FUNCTION_BLOCK FB_HomingProcessor
VAR_IN_OUT
	J1, J2, J3, J4, J5, J6: AXIS_REF;
	AxisGroup: AXIS_GROUP_REF_SM3;
	GroupHandler: FB_GroupHandler;
	Controller: FB_Controller;
END_VAR

VAR_INPUT
	J1_Limit, J2_Limit, J3_Limit, J4_Limit, J5_Limit, J6_Limit: BOOL;
	Enable: BOOL;
	Reset: BOOL;
	StoredPositions: REFERENCE TO ARRAY[GVL.POS_ARR_BEG..GVL.POS_ARR_END] OF DUT_StoredPosition;
	VisionRegisters: REFERENCE TO ARRAY[GVL.VIS_ARR_BEG..GVL.VIS_ARR_END] OF DUT_VisionRegister;
	Flags: REFERENCE TO ARRAY[GVL.FLG_ARR_BEG..GVL.FLG_ARR_END] OF DUT_Flags;
END_VAR
VAR_OUTPUT
	Done: BOOL;
	Busy: BOOL;
	Error: BOOL;
	ErrorID: UDINT;
END_VAR
VAR
	_ExecuteRtrig: R_TRIG;
	_ExecuteFtrig: F_TRIG;
	_ResetRtrig: R_TRIG;
	_ErrorRtrig: R_TRIG;
	
	_SequenceMain: INT;
	_StartHoming: BOOL;
	
	_SMC_Homing_J1, _SMC_Homing_J2, _SMC_Homing_J3: MC_Home;
	_SMC_Homing_J4, _SMC_Homing_J5, _SMC_Homing_J6: MC_Home;
    _ST_HomingOptions_J1,_ST_HomingOptions_J2,_ST_HomingOptions_J3: ST_HomingOptions;
    _ST_HomingOptions_J4,_ST_HomingOptions_J5,_ST_HomingOptions_J6: ST_HomingOptions;
	
	_MC_SetPosition_J1, _MC_SetPosition_J2, _MC_SetPosition_J3: MC_SetPosition;
	_MC_SetPosition_J4, _MC_SetPosition_J5, _MC_SetPosition_J6: MC_SetPosition;
    _ST_SetPositionsOptions_J1,_ST_SetPositionsOptions_J2,_ST_SetPositionsOptions_J3: ST_SetPositionOptions;
    _ST_SetPositionsOptions_J4,_ST_SetPositionsOptions_J5,_ST_SetPositionsOptions_J6: ST_SetPositionOptions;
	
	_HomingVelocityFast: LREAL:= 10.0;
	_HomingVelocitySlow: LREAL:= 5.0;
	_HomingVelocitySlowSlow: LREAL:= 1.0;
	_HomingAcceleration: LREAL:= 1000.0;
	_HomingJerk: LREAL:= 10000.0;
	
	_MoveToPose: BOOL;
	_MoveCommand: ST_MoveCmd;
	_MoveCommandProcessor: MoveCmdProcessor;
	
	_i, _j, _k: INT;
	_FirstScan: BOOL:=TRUE;
END_VAR

VAR CONSTANT
	STEP_DONE: 					INT := 9999;
	STEP_IDLE: 					INT := 0000;
	STEP_GROUP_ENABLE: 			INT := 0030;
	STEP_WAIT_ENABLE: 			INT := 0035;
	STEP_FAST_HOME_G1:			INT := 0040;
	STEP_WAIT_FAST_HOME_G1:		INT := 0045;
	STEP_SLOW_HOME_G1:			INT := 0050;
	STEP_WAIT_SLOW_HOME_G1:		INT := 0055;
	
	STEP_FAST_HOME_G2:			INT := 0060;
	STEP_WAIT_FAST_HOME_G2:		INT := 0065;
	STEP_SLOW_HOME_G2:			INT := 0070;
	STEP_WAIT_SLOW_HOME_G2:		INT := 0075;
	
	STEP_FAST_HOME_G3:			INT := 0080;
	STEP_WAIT_FAST_HOME_G3:		INT := 0085;
	STEP_SLOW_HOME_G3:			INT := 0090;
	STEP_WAIT_SLOW_HOME_G3:		INT := 0095;
	
	STEP_MOVE_TO_POSE:			INT := 1000;
	STEP_WAIT_MOVE_TO_POSE:		INT := 1010;
	STEP_WAIT_POSE_DONE:		INT := 1020;
END_VAR

_ExecuteRtrig(CLK:=);
_ExecuteFtrig(CLK:=);
_ResetRtrig(CLK:=Reset);

IF _FirstScan THEN
	//
END_IF

CASE _SequenceMain OF
	STEP_DONE: // done
		Busy := FALSE;
		Done := TRUE;
		_MoveCommandProcessor.M_Home();
		_SequenceMain := STEP_IDLE;
		
		_SMC_Homing_J1.Execute := FALSE;
		_SMC_Homing_J2.Execute := FALSE;
		_SMC_Homing_J3.Execute := FALSE;
		_SMC_Homing_J4.Execute := FALSE;
		_SMC_Homing_J5.Execute := FALSE;
		_SMC_Homing_J6.Execute := FALSE;
		(*J1.bSWLimitEnable := TRUE;
		J2.bSWLimitEnable := TRUE;
		J3.bSWLimitEnable := TRUE;
		J4.bSWLimitEnable := TRUE;
		J5.bSWLimitEnable := TRUE;
		J6.bSWLimitEnable := TRUE;*)
		
	STEP_IDLE: // IDLE
		IF _StartHoming AND Enable THEN
			_StartHoming := FALSE;
			Busy := TRUE;
			Done := FALSE;
			_SequenceMain := STEP_GROUP_ENABLE;
			Flags[GVL.HOME_COMPLETE].Value := FALSE;
		END_IF
		
	STEP_GROUP_ENABLE:
		IF GroupHandler.M_EnableGroup() THEN
			_SequenceMain := STEP_WAIT_ENABLE;
		ELSE
			_SequenceMain := STEP_DONE;
			Error := TRUE;
			ErrorID := GroupHandler.ErrorID;
		END_IF
		
	STEP_WAIT_ENABLE:
		// TODO add timeout timer here
		IF GroupHandler.P_GroupEnabled THEN
			_SequenceMain := STEP_FAST_HOME_G1;
		END_IF;
		
	STEP_FAST_HOME_G1:	
		_SMC_Homing_J1.Execute := TRUE;
		_SMC_Homing_J2.Execute := TRUE;
		_SMC_Homing_J3.Execute := TRUE;
		//_SMC_Homing_J1.bReturnToZero := FALSE;
		//_SMC_Homing_J2.bReturnToZero := FALSE;
		//_SMC_Homing_J3.bReturnToZero := FALSE;
		_SMC_Homing_J1.Options.SearchVelocity := _HomingVelocitySlow;
		_SMC_Homing_J2.Options.SearchVelocity := _HomingVelocitySlow;
		_SMC_Homing_J3.Options.SearchVelocity := _HomingVelocitySlow;
		//J1.bSWLimitEnable := FALSE;
		//J2.bSWLimitEnable := FALSE;
		//J3.bSWLimitEnable := FALSE;
		_SequenceMain := STEP_WAIT_FAST_HOME_G1;
		
	STEP_WAIT_FAST_HOME_G1: // wait fast home group 1
		IF _SMC_Homing_J1.Done
			AND _SMC_Homing_J2.Done
			AND _SMC_Homing_J3.Done THEN
				_SMC_Homing_J1.Execute := FALSE;
				_SMC_Homing_J2.Execute := FALSE;
				_SMC_Homing_J3.Execute := FALSE;
				_SequenceMain := STEP_SLOW_HOME_G1;
		END_IF
		
	STEP_SLOW_HOME_G1: // slow home group 1
		_SMC_Homing_J1.Execute := TRUE;
		_SMC_Homing_J2.Execute := TRUE;
		_SMC_Homing_J3.Execute := TRUE;
		//_SMC_Homing_J1.bReturnToZero := TRUE;
		//_SMC_Homing_J2.bReturnToZero := TRUE;
		//_SMC_Homing_J3.bReturnToZero := TRUE;
		_SMC_Homing_J1.Options.SearchVelocity := _HomingVelocitySlowSlow;
		_SMC_Homing_J2.Options.SearchVelocity := _HomingVelocitySlowSlow;
		_SMC_Homing_J3.Options.SearchVelocity := _HomingVelocitySlowSlow;
		_SequenceMain := STEP_WAIT_SLOW_HOME_G1;
		
	STEP_WAIT_SLOW_HOME_G1:
		IF _SMC_Homing_J1.Done
			AND _SMC_Homing_J2.Done
			AND _SMC_Homing_J3.Done THEN
				_SMC_Homing_J1.Execute := FALSE;
				_SMC_Homing_J2.Execute := FALSE;
				_SMC_Homing_J3.Execute := FALSE;
				_SequenceMain := STEP_FAST_HOME_G2;
		END_IF
		
	STEP_FAST_HOME_G2:		
		_SMC_Homing_J4.Execute := TRUE;
		_SMC_Homing_J5.Execute := TRUE;
		//_SMC_Homing_J4.bReturnToZero := FALSE;
		//_SMC_Homing_J5.bReturnToZero := FALSE;
		_SMC_Homing_J4.Options.SearchVelocity := _HomingVelocitySlow;
		_SMC_Homing_J5.Options.SearchVelocity := _HomingVelocitySlow;
		//J4.bSWLimitEnable := FALSE;
		//J5.bSWLimitEnable := FALSE;
		_SequenceMain := STEP_WAIT_FAST_HOME_G2;
		
	STEP_WAIT_FAST_HOME_G2:
		IF _SMC_Homing_J4.Done
			AND _SMC_Homing_J5.Done THEN
				_SMC_Homing_J4.Execute := FALSE;
				_SMC_Homing_J5.Execute := FALSE;
				_SequenceMain := STEP_SLOW_HOME_G2;
		END_IF
		
	STEP_SLOW_HOME_G2:
		_SMC_Homing_J4.Execute := TRUE;
		_SMC_Homing_J5.Execute := TRUE;
		//_SMC_Homing_J4.bReturnToZero := TRUE;
		//_SMC_Homing_J5.bReturnToZero := TRUE;
		_SMC_Homing_J4.Options.SearchVelocity := _HomingVelocitySlowSlow;
		_SMC_Homing_J5.Options.SearchVelocity := _HomingVelocitySlowSlow;
		_SequenceMain := STEP_WAIT_SLOW_HOME_G2;
		
	STEP_WAIT_SLOW_HOME_G2:
		IF _SMC_Homing_J4.Done
			AND _SMC_Homing_J5.Done THEN
				_SMC_Homing_J4.Execute := FALSE;
				_SMC_Homing_J5.Execute := FALSE;
				_SequenceMain := STEP_FAST_HOME_G3;
		END_IF
		
	STEP_FAST_HOME_G3:
		_SMC_Homing_J6.Execute := TRUE;
		//_SMC_Homing_J6.bReturnToZero := FALSE;
		_SMC_Homing_J6.Options.SearchVelocity := _HomingVelocitySlow;
		//J6.bSWLimitEnable := FALSE;
		_SequenceMain := STEP_WAIT_FAST_HOME_G3;
		
	STEP_WAIT_FAST_HOME_G3:
		IF _SMC_Homing_J6.Done THEN
			_SMC_Homing_J6.Execute := FALSE;
			_SequenceMain := STEP_SLOW_HOME_G3;
		END_IF
		
	STEP_SLOW_HOME_G3:
		_SMC_Homing_J6.Execute := TRUE;
		//_SMC_Homing_J6.bReturnToZero := TRUE;
		_SMC_Homing_J6.Options.SearchVelocity := _HomingVelocitySlowSlow;
		_SequenceMain := STEP_WAIT_SLOW_HOME_G3;
		
	STEP_WAIT_SLOW_HOME_G3:
		IF _SMC_Homing_J6.Done THEN
			_SMC_Homing_J6.Execute := FALSE;
			Flags[GVL.HOME_COMPLETE].Value := TRUE;
			IF NOT Flags[GVL.HOM_TO_POSE_IDX].Value THEN
				_SequenceMain := STEP_DONE;
			ELSE
				_SequenceMain := STEP_MOVE_TO_POSE;
			END_IF
		END_IF;
		
	STEP_MOVE_TO_POSE:
		_MoveToPose := TRUE;
		_SequenceMain := STEP_WAIT_MOVE_TO_POSE;
	
	STEP_WAIT_MOVE_TO_POSE:
		IF _MoveCommandProcessor.ItfUnitMode.CurrentState <> PACK_ML.State.Idle THEN
			_SequenceMain := STEP_WAIT_POSE_DONE;
		END_IF
		
	STEP_WAIT_POSE_DONE:
		IF _MoveCommandProcessor.ItfUnitMode.CurrentState = PACK_ML.State.Idle THEN
			_SequenceMain := STEP_DONE;
		END_IF
	
END_CASE

_M_HandlePose();

//
IF _ResetRtrig.Q AND Error THEN
	Error := FALSE;
	ErrorID := 0;
	_SequenceMain := STEP_DONE;
	GroupHandler.M_ResetGroup();
	_MoveCommandProcessor.M_Home();
END_IF

//
_ErrorRtrig(CLK:=GroupHandler.Error
				OR _SMC_Homing_J1.Error
				OR _SMC_Homing_J2.Error
				OR _SMC_Homing_J3.Error
				OR _SMC_Homing_J4.Error
				OR _SMC_Homing_J5.Error
				OR _SMC_Homing_J6.Error
				OR _MoveCommandProcessor.Error);			
IF _ErrorRtrig.Q THEN
	Error := TRUE;
	IF GroupHandler.Error THEN
		ErrorID := GroupHandler.ErrorID;
	ELSIF _SMC_Homing_J1.Error THEN
		ErrorID := _SMC_Homing_J1.ErrorID;
	ELSIF _SMC_Homing_J2.Error THEN
		ErrorID := _SMC_Homing_J2.ErrorID;
	ELSIF _SMC_Homing_J3.Error THEN
		ErrorID := _SMC_Homing_J3.ErrorID;
	ELSIF _SMC_Homing_J4.Error THEN
		ErrorID := _SMC_Homing_J4.ErrorID;
	ELSIF _SMC_Homing_J5.Error THEN
		ErrorID := _SMC_Homing_J5.ErrorID;
	ELSIF _SMC_Homing_J6.Error THEN
		ErrorID := _SMC_Homing_J6.ErrorID;
	ELSIF _MoveCommandProcessor.Error THEN
		// TODO need to rework how error messages are handled (globally)
		// if the move command processor has an error, we dont know what it is.
	END_IF
END_IF

// TODO make search direction configurable for any robot
//
_ST_HomingOptions_J1.SearchDirection := MC_Negative_Direction;
_SMC_Homing_J1(
	Axis:= J1, 
	Execute:= , 
	Position:= StoredPositions[GVL.HOM_POS_IDX].Position.X, 
	HomingMode:= MC_HomingMode.MC_DefaultHoming, 
	BufferMode:= , 
	Options:= _ST_HomingOptions_J1, 
	bCalibrationCam:= , 
	Done=> , 
	Busy=> , 
	Active=> , 
	CommandAborted=> , 
	Error=> , 
	ErrorID=> );
(*_SMC_Homing_J1(
	Axis:=J1 , 
	Execute:= ,
	Position:= StoredPositions[GVL.HOM_POS_IDX].Position.X, 
	fVelocitySlow:= , 
	fVelocityFast:= _HomingVelocityFast, 
	fAcceleration:= _HomingAcceleration, 
	fDeceleration:= _HomingAcceleration, 
	fJerk:= _HomingJerk, 
	nDirection:= MC_direction.negative, 
	bReferenceSwitch:= NOT J1_Limit, 
	fSignalDelay:= , 
	nHomingMode:= , 
	bReturnToZero:= , 
	bIndexOccured:= , 
	fIndexPosition:= , 
	bIgnoreHWLimit:= TRUE, 
	bDone=> , 
	bBusy=> , 
	bCommandAborted=> , 
	bError=> , 
	nErrorID=> , 
	bStartLatchingIndex=> );
	
_SMC_Homing_J2(
	Axis:=J2 , 
	bExecute:= , 
	fHomePosition:= StoredPositions[GVL.HOM_POS_IDX].Position.Y,  
	fVelocitySlow:= , 
	fVelocityFast:= _HomingVelocityFast, 
	fAcceleration:= _HomingAcceleration, 
	fDeceleration:= _HomingAcceleration,
	fJerk:= _HomingJerk, 
	nDirection:= MC_Direction.negative, 
	bReferenceSwitch:= NOT J2_Limit, 
	fSignalDelay:= , 
	nHomingMode:= , 
	bReturnToZero:= , 
	bIndexOccured:= , 
	fIndexPosition:= , 
	bIgnoreHWLimit:= TRUE, 
	bDone=> , 
	bBusy=> , 
	bCommandAborted=> , 
	bError=> , 
	nErrorID=> , 
	bStartLatchingIndex=> );
	
_SMC_Homing_J3(
	Axis:=J3 , 
	bExecute:= , 
	fHomePosition:= StoredPositions[GVL.HOM_POS_IDX].Position.Z, 
	fVelocitySlow:= , 
	fVelocityFast:= _HomingVelocityFast, 
	fAcceleration:= _HomingAcceleration, 
	fDeceleration:= _HomingAcceleration,
	fJerk:= _HomingJerk, 
	nDirection:= MC_Direction.positive, 
	bReferenceSwitch:= NOT J3_Limit, 
	fSignalDelay:= , 
	nHomingMode:= , 
	bReturnToZero:= , 
	bIndexOccured:= , 
	fIndexPosition:= , 
	bIgnoreHWLimit:= TRUE, 
	bDone=> , 
	bBusy=> , 
	bCommandAborted=> , 
	bError=> , 
	nErrorID=> , 
	bStartLatchingIndex=> );
	
_SMC_Homing_J4(
	Axis:=J4 , 
	bExecute:= ,
	fHomePosition:= StoredPositions[GVL.HOM_POS_IDX].Position.A, 
	fVelocitySlow:= , 
	fVelocityFast:= _HomingVelocityFast, 
	fAcceleration:= _HomingAcceleration, 
	fDeceleration:= _HomingAcceleration,
	fJerk:= _HomingJerk, 
	nDirection:= MC_Direction.positive, 
	bReferenceSwitch:= NOT J4_Limit, 
	fSignalDelay:= , 
	nHomingMode:= , 
	bReturnToZero:= , 
	bIndexOccured:= , 
	fIndexPosition:= , 
	bIgnoreHWLimit:= TRUE, 
	bDone=> , 
	bBusy=> , 
	bCommandAborted=> , 
	bError=> , 
	nErrorID=> , 
	bStartLatchingIndex=> );
	
_SMC_Homing_J5(
	Axis:=J5 , 
	bExecute:= , 
	fHomePosition:= StoredPositions[GVL.HOM_POS_IDX].Position.B,  
	fVelocitySlow:= , 
	fVelocityFast:= _HomingVelocityFast, 
	fAcceleration:= _HomingAcceleration, 
	fDeceleration:= _HomingAcceleration,
	fJerk:= _HomingJerk, 
	nDirection:= MC_Direction.positive, 
	bReferenceSwitch:= NOT J5_Limit, 
	fSignalDelay:= , 
	nHomingMode:= , 
	bReturnToZero:= , 
	bIndexOccured:= , 
	fIndexPosition:= , 
	bIgnoreHWLimit:= TRUE, 
	bDone=> , 
	bBusy=> , 
	bCommandAborted=> , 
	bError=> , 
	nErrorID=> , 
	bStartLatchingIndex=> );
	
_SMC_Homing_J6(
	Axis:=J6 , 
	bExecute:= , 
	fHomePosition:= StoredPositions[GVL.HOM_POS_IDX].Position.C, 
	fVelocitySlow:= , 
	fVelocityFast:= _HomingVelocityFast, 
	fAcceleration:= _HomingAcceleration, 
	fDeceleration:= _HomingAcceleration,
	fJerk:= _HomingJerk, 
	nDirection:= MC_Direction.negative, 
	bReferenceSwitch:= NOT J6_Limit, 
	fSignalDelay:= , 
	nHomingMode:= , 
	bReturnToZero:= , 
	bIndexOccured:= , 
	fIndexPosition:= , 
	bIgnoreHWLimit:= TRUE, 
	bDone=> , 
	bBusy=> , 
	bCommandAborted=> , 
	bError=> , 
	nErrorID=> , 
	bStartLatchingIndex=> );
    *)
	
//
_ST_SetPositionsOptions_J1.ClearPositionLag := TRUE;
_MC_SetPosition_J1(
	Axis:= J1, 
	Execute:= _MC_SetPosition_J1.Execute AND NOT _MC_SetPosition_J1.Done AND NOT _MC_SetPosition_J1.Error, 
	Position:= 0.0, 
	Mode:= FALSE, // true=relative false=absolute
    Options:= _ST_SetPositionsOptions_J1,
	Done=> , 
	Busy=> , 
	Error=> , 
	ErrorID=> );
_ST_SetPositionsOptions_J2.ClearPositionLag := TRUE;
_MC_SetPosition_J2(
	Axis:= J2, 
	Execute:= _MC_SetPosition_J2.Execute AND NOT _MC_SetPosition_J2.Done AND NOT _MC_SetPosition_J2.Error, 
	Position:= 0.0, 
	Mode:= FALSE, // true=relative false=absolute
    Options:= _ST_SetPositionsOptions_J2,
	Done=> , 
	Busy=> , 
	Error=> , 
	ErrorID=> );
_ST_SetPositionsOptions_J3.ClearPositionLag := TRUE;
_MC_SetPosition_J3(
	Axis:= J3, 
	Execute:= _MC_SetPosition_J3.Execute AND NOT _MC_SetPosition_J3.Done AND NOT _MC_SetPosition_J3.Error, 
	Position:= 0.0, 
	Mode:= FALSE, // true=relative false=absolute
    Options:= _ST_SetPositionsOptions_J3,
	Done=> , 
	Busy=> , 
	Error=> , 
	ErrorID=> );
_ST_SetPositionsOptions_J4.ClearPositionLag := TRUE;
_MC_SetPosition_J4(
	Axis:= J4, 
	Execute:= _MC_SetPosition_J4.Execute AND NOT _MC_SetPosition_J4.Done AND NOT _MC_SetPosition_J4.Error, 
	Position:= 0.0, 
	Mode:= FALSE, // true=relative false=absolute
    Options:= _ST_SetPositionsOptions_J4,
	Done=> , 
	Busy=> , 
	Error=> , 
	ErrorID=> );
_ST_SetPositionsOptions_J5.ClearPositionLag := TRUE;
_MC_SetPosition_J5(
	Axis:= J5, 
	Execute:= _MC_SetPosition_J5.Execute AND NOT _MC_SetPosition_J5.Done AND NOT _MC_SetPosition_J5.Error, 
	Position:= 0.0, 
	Mode:= FALSE, // true=relative false=absolute
    Options:= _ST_SetPositionsOptions_J5,
	Done=> , 
	Busy=> , 
	Error=> , 
	ErrorID=> );
_ST_SetPositionsOptions_J6.ClearPositionLag := TRUE;
_MC_SetPosition_J6(
	Axis:= J6, 
	Execute:= _MC_SetPosition_J6.Execute AND NOT _MC_SetPosition_J6.Done AND NOT _MC_SetPosition_J6.Error, 
	Position:= 0.0, 
	Mode:= FALSE, // true=relative false=absolute
    Options:= _ST_SetPositionsOptions_J6,
	Done=> , 
	Busy=> , 
	Error=> , 
	ErrorID=> );

METHOD PRIVATE _M_HandlePose : BOOL
VAR
	_MoveCommand: ST_MoveCmd;
	_PoseSpeed: LREAL := 20.0;
END_VAR
IF _MoveToPose THEN
	_MoveToPose:= FALSE;
	//
	IF GVL.PowerOn 
		AND_THEN Flags[GVL.HOME_COMPLETE].Value
		AND_THEN NOT _MoveCommandProcessor.Busy
		AND_THEN NOT _MoveCommandProcessor.Error THEN
			//
			_MoveCommand.MoveType 			:= DUT_Command_MoveType.DirectMove;
			_MoveCommand.PositionType 		:= DUT_Command_PositionType.AbsolutePosition;
			_MoveCommand.CoordinateType 	:= DUT_Command_CoordinateType.Literal;
			_MoveCommand.Speed 				:= _PoseSpeed;
			_MoveCommand.CoordSystem 		:= SMC_COORD_SYSTEM.ACS;
			_MoveCommand.CoordRef 			:= StoredPositions[GVL.POSE_2_IDX].Position;
			//
			_MoveCommandProcessor.Command := BuildMoveCmd(_MoveCommand);
			_MoveCommandProcessor.M_Start();
	END_IF;
END_IF

_MoveCommandProcessor(
	StoredPositions:= StoredPositions,
	VisionRegisters:= VisionRegisters,
	Flags:= Flags,
	AxisGroup:= AxisGroup, 
	GroupHandler:= GroupHandler,
	Velocity:= StoredPositions[GVL.SPEEDS_IDX].Position.X, 
	VelFactor:= StoredPositions[GVL.SPEEDS_IDX].Position.A,
	Acceleration:= StoredPositions[GVL.SPEEDS_IDX].Position.Y, 
	AccFactor:= StoredPositions[GVL.SPEEDS_IDX].Position.B,
	Jerk:= StoredPositions[GVL.SPEEDS_IDX].Position.Z,
	JerkFactor:= StoredPositions[GVL.SPEEDS_IDX].Position.C, 
	Position=> ,
	ItfUnitMode=> , 
	Error=> );
END_METHOD

METHOD M_SetHome : BOOL

// adjust all the persistent variables to take on the calibrated values
StoredPositions[GVL.HOM_POS_IDX].Position.X := F_HomeOffsetCalc(	CurrentOffset:= PersistentVars.StoredPositions[GVL.HOM_POS_IDX].Position.X, 
																				CurrentPosition:= J1.fActPosition, 
																				HomeSearchDirection:= _SMC_Homing_J1.nDirection);

StoredPositions[GVL.HOM_POS_IDX].Position.Y := F_HomeOffsetCalc(	CurrentOffset:= PersistentVars.StoredPositions[GVL.HOM_POS_IDX].Position.Y, 
																				CurrentPosition:= J2.fActPosition, 
																				HomeSearchDirection:= _SMC_Homing_J2.nDirection);

StoredPositions[GVL.HOM_POS_IDX].Position.Z := F_HomeOffsetCalc(	CurrentOffset:= PersistentVars.StoredPositions[GVL.HOM_POS_IDX].Position.Z, 
																				CurrentPosition:= J3.fActPosition, 
																				HomeSearchDirection:= _SMC_Homing_J3.nDirection);

StoredPositions[GVL.HOM_POS_IDX].Position.A := F_HomeOffsetCalc(	CurrentOffset:= PersistentVars.StoredPositions[GVL.HOM_POS_IDX].Position.A, 
																				CurrentPosition:= J4.fActPosition, 
																				HomeSearchDirection:= _SMC_Homing_J4.nDirection);

StoredPositions[GVL.HOM_POS_IDX].Position.B := F_HomeOffsetCalc(	CurrentOffset:= PersistentVars.StoredPositions[GVL.HOM_POS_IDX].Position.B, 
																				CurrentPosition:= J5.fActPosition, 
																				HomeSearchDirection:= _SMC_Homing_J5.nDirection);

StoredPositions[GVL.HOM_POS_IDX].Position.C := F_HomeOffsetCalc(	CurrentOffset:= PersistentVars.StoredPositions[GVL.HOM_POS_IDX].Position.C, 
																				CurrentPosition:= J6.fActPosition, 
																				HomeSearchDirection:= _SMC_Homing_J6.nDirection);

// this isnt totally needed but will calibrate the current session without the need to rehome
_MC_SetPosition_J1.Execute:=TRUE;
_MC_SetPosition_J2.Execute:=TRUE;
_MC_SetPosition_J3.Execute:=TRUE;
_MC_SetPosition_J4.Execute:=TRUE;
_MC_SetPosition_J5.Execute:=TRUE;
_MC_SetPosition_J6.Execute:=TRUE;
END_METHOD

METHOD M_StartHoming : BOOL
IF _SequenceMain = STEP_IDLE THEN
	M_StartHoming := TRUE;
	_StartHoming := TRUE;
ELSE
	M_StartHoming := FALSE;
END_IF
END_METHOD

END_FUNCTION_BLOCK

(* stored: Version 1.1.0.1
   POU FB_HomingProcessor: Id {6c30ff35-bc31-4ed8-ab4a-320ad080dc49}, SpecialFunc None
   Method _M_HandlePose: Id {8dbad245-108d-44dc-844d-47ebe55e9287}
   Method M_SetHome: Id {ac8ad3ff-e2e3-4571-99f3-004f0df0c316}
   Method M_StartHoming: Id {1ff714ca-aba4-448a-bc01-bf0eab578f27} *)
